{attribute 'GeneratedUsingTerminal: EP1816-0008-0016'}
{attribute addProperty BoxType "EP1816-0008-0016"}
{attribute addProperty Description "EP1816-0008 16 Ch. Dig. Input 24V, 10µs, D-SUB25"}
{attribute addProperty Physics "YY"}
{attribute addProperty Id "DO_Inputs_Channel_1AT %I*DO_Inputs_Channel_CC4551489DO_Inputs_Channel_2AT %I*DO_Inputs_Channel_CC4551489WcStateAT %I*WcState_9091E0EB2InfoDataAT %I*InfoData_32EB74EA10"}
{attribute addProperty CRC "64520457"}
{attribute addProperty Size "30"}
TYPE EP1816_03D88109 EXTENDS EtcSlaveBoxBase_77A0E4A7 :
STRUCT
	{attribute addProperty Name "DO_Inputs_Channel_1"}
	DO_Inputs_Channel_1 : DO_Inputs_Channel_CC455148;
	{attribute addProperty Name "DO_Inputs_Channel_2"}
	DO_Inputs_Channel_2 : DO_Inputs_Channel_CC455148;
	{attribute addProperty Name "WcState"}
	WcState : WcState_9091E0EB;
	{attribute addProperty Name "InfoData"}
	InfoData : InfoData_32EB74EA;
END_STRUCT
END_TYPE

(* stored: Version 1.2.0.0, ProductVersion 3.1.4024.9
   DUT EP1816_03D88109: Id {a7acd4c8-7565-41d3-93b8-e1e65fbeb205} *)
